// TIA Portal V16 export
// export: Created 2024-12-03T15:41:45.0415446Z, ExportSetting WithReadOnly, DisplayName Totally Integrated Automation Portal, DisplayVersion V16 Update 6, DisplayName TIA Portal Version Control Interface, DisplayVersion V16 Update 2, DisplayName TIA Portal Openness, DisplayVersion V16 Update 6, DisplayName TIA Portal Teamcenter Gateway, DisplayVersion V16, DisplayName SINAMICS Startdrive Advanced, DisplayVersion V16 Update 5, DisplayName SINAMICS Startdrive G130, G150, S120, S150, SINAMICS MV, S210, DisplayVersion V16 Update 5, DisplayName SINAMICS Startdrive G110M, G120, G120C, G120D, G120P, G115D, DisplayVersion V16 Update 5, DisplayName STEP 7 Professional, DisplayVersion V16 Update 6, DisplayName STEP 7 Safety, DisplayVersion V16, DisplayName WinCC Advanced / Unified PC, DisplayVersion V16 Update 6
TYPE "ConveyLinxAlarms"
// stored: CreationDate 2021-07-13T07:41:36.2278727Z, InterfaceModifiedDate 2020-02-08T17:11:40.2341278Z, IsConsistent true, LibraryConformanceStatus The object is library-conformant., ModifiedDate 2021-03-27T07:36:47.6287659Z
   STRUCT
      Overheat { ExternalVisible := 'False'} : "HmiAlarm";   // The MDR 's temperature has exceeded 105 degrees Celsius
      ShortCircuit { ExternalVisible := 'False'} : "HmiAlarm";   // There is a short circuit on the MDR
      MDRNotConnected { ExternalVisible := 'False'} : "HmiAlarm";   // The MDR is not connected
      Overload { ExternalVisible := 'False'} : "HmiAlarm";   // The MDR has been overloaded - this means its speed is less than 10% of the selected speed
      Stalled { ExternalVisible := 'False'} : "HmiAlarm";   // The MDR has stalled
      MDRBadHall { ExternalVisible := 'False'} : "HmiAlarm";   // The MDR has a Hall Efect Sensor error
      OverVoltage { ExternalVisible := 'False'} : "HmiAlarm";   // The sum of the module power supply voltage + the MDR-generated voltage has exceeded 30 volts
      LowVoltage { ExternalVisible := 'False'} : "HmiAlarm";   // Module power supply is less than 18 Volts
      NotConnected : "HmiAlarm";   // The module is not connected
      ConnectionNotOK : "HmiAlarm";   // The Ethernet connections are not ok .
      AnyErrorActive : "HmiAlarm";   // Any Error is active
      JamError : "HmiAlarm";   // Jam Error
      SensorLowGain : "HmiAlarm";   // Sensor Low gain
      Status_1 : Word;   // lsb => 0 overheat | 1 spare | 2 shortcircuit | 3 mdrn not connected | 4 overload | 5 stalled | 6 bad hall | 7 spare | 8 over voltage | 9 low voltage | 10 not connected | 11 conneciton nok | 12 anyError | 13 jam error | 14 Sensor log gain
   END_STRUCT;
END_TYPE
